"WR_REC"	SFC 58	SFC 58	// WRITE DATA RECORD
"RD_REC"	SFC 59	SFC 59	// READ A DATA RECORD
"TIME_TCK"	SFC 64	SFC 64	// READ THE SYSTEM TIME
"GEO_LOG"	SFC 70	SFC 70	// DETERMINE LOGICAL ADDRESS
"READ_DBL"	SFC 83	SFC 83	// READ DATA BLOCK OUT OF LOAD MEMORY
"WRIT_DBL"	SFC 84	SFC 84	// WRITE DATA BLOCK IN LOAD MEMORY
"DEL_SI"	SFC 106	SFC 106	// Deleting Dynamically Assigned System Instances
"ALARM_DQ"	SFC 107	SFC 107	// Creating Acknowledgeable Block-related Message
"ALARM_D"	SFC 108	SFC 108	// Creating Acknowledged Block-related Message
"LIEN_SEC"	UDT 1507	UDT 1507	// TABLE COMMUNE AUX BF_ZONE_PORTE1, BF_ZONE_RSEC1, BF_ZONE_MODE_IHM, BF_ZONE_AIR
"MOT_FONC_DPL"	UDT 1866	UDT 1866
"LIEN_PUP"	UDT 1988	UDT 1988	// Gestion des Modes et des pupitres de cde manu de la  zone (BF_ZONE_MODE_IHM)
"LIEN_ILOT"	UDT 2004	UDT 2004	// INFO CONTROL LINKED TO THE FACILITY (BF_ILOT)
"MOT_FONC_MP"	UDT 2041	UDT 2041	// INFO CONTROL OF A MOVEMENT (BF_MOUVMP1)
"MOT_FONC"	UDT 2042	UDT 2042
"VAT_SIPTOL"	VAT 1	
"VAT_TALOA0"	VAT 2	
"VAT_BASE DE DADOS"	VAT 3	
"Z1T_TEMPOS"	VAT 4	
"Z2T_TEMPOS"	VAT 5	
"VAT_6"	VAT 6	
"acompanhamento zona 8"	VAT 7		// teste tucker
"TOMAS"	VAT 8	
"W0"	VAT 9	
"VAT_Z1_BOT_EMER"	VAT 10	
"VAT_Z2_BOT_EMER"	VAT 11		// BOTAO_DE_EMERGENCIA
"VAT_Z1_VALIDAÇÃO"	VAT 12	
"VAT_CDIV_2"	VAT 13	
"VAT_Z2_VALIDAÇÃO"	VAT 14	
"ELEV_CARREGAMENTO"	VAT 15	
"ELEV_DESCARREGAMENTO"	VAT 16	
"VAT_17"	VAT 17	
"TESTE_MODO_DEGR"	VAT 18	
"VAT_SIPTOL_TOM"	VAT 19	
"mostrar IIT"	VAT 20	
"tab_iit_2"	VAT 21	
"VAT_22"	VAT 22	
"afficher"	VAT 23	
END_SYMBOL_TABLE
